{region '#Template'}
	{attribute 'Version' := '1.0.0.0'}
	{attribute 'Tags' := '"LCID": "1031", "Text": "AC, General, night cooling"'}
	{attribute 'Tags' := '"LCID": "1033", "Text": "AC, General, night cooling"'}
	{attribute 'Description' := '"LCID": "1031", "Text": "Nachtkühlung"'}
	{attribute 'Description' := '"LCID": "1033", "Text": "night cooling"'}
{endregion}
FUNCTION_BLOCK FB_BA_AC_SumNgtCol EXTENDS FB_BA_View
VAR_INPUT
	fTRm					: REAL;
	fSpRm					: REAL;
	fTWth					: REAL;		
END_VAR
VAR_OUTPUT
	bQ						: BOOL;
END_VAR
VAR_INPUT CONSTANT
	WthTLoLmt				: FB_BA_AV_Op;	
	RmTHys					: FB_BA_AV_Op;	
	SwiOnDiffT				: FB_BA_AV_Op;	
	SwiOffDiffT				: FB_BA_AV_Op;	
	Q						: FB_BA_BV_Op;																					
	Sched					: FB_BA_SchedM;
END_VAR
VAR
	NgtColFnct				: FB_BA_NgtCol;
END_VAR

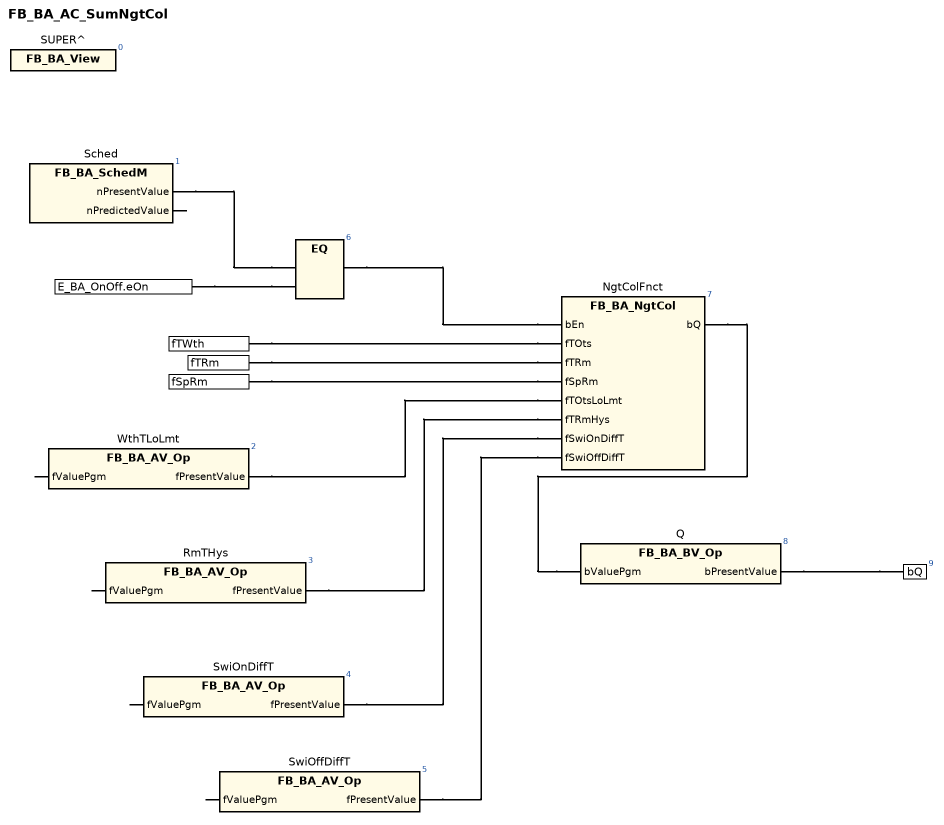
SUPER^(); // FB_BA_View
Sched(); // FB_BA_SchedM
WthTLoLmt(); // FB_BA_AV_Op
RmTHys(); // FB_BA_AV_Op
SwiOnDiffT(); // FB_BA_AV_Op
SwiOffDiffT(); // FB_BA_AV_Op
NgtColFnct(
    bEn := Sched.nPresentValue = E_BA_OnOff.eOn,
    fTOts := fTWth,
    fTRm := fTRm,
    fSpRm := fSpRm,
    fTOtsLoLmt := WthTLoLmt.fPresentValue,
    fTRmHys := RmTHys.fPresentValue,
    fSwiOnDiffT := SwiOnDiffT.fPresentValue,
    fSwiOffDiffT := SwiOffDiffT.fPresentValue); // FB_BA_NgtCol
Q(bValuePgm := NgtColFnct.bQ); // FB_BA_BV_Op
bQ := Q.bPresentValue;

METHOD FB_init : BOOL
VAR_INPUT
	bInitRetains : BOOL; // if TRUE, the retain variables are initialized (warm start / cold start)
	bInCopyCode : BOOL;  // if TRUE, the instance afterwards gets moved into the copy code (online change)
END_VAR
WthTLoLmt.iParent			:= THIS^;
WthTLoLmt.iLabel			:= LblCmpAC.General_SumNgtCol_WthTLoLmt;			
WthTLoLmt.sObjectName		:= '{Idx=01}';								 	 
WthTLoLmt.eUnit				:= E_BA_Unit.eTemperature_DegreesCelsius;  
WthTLoLmt.fValueRm			:= 9.0;

RmTHys.iParent				:= THIS^;
RmTHys.iLabel				:= LblCmpAC.General_SumNgtCol_RmTHys;			
RmTHys.sObjectName			:= '{Idx=01}';								 	 
RmTHys.eUnit				:= E_BA_Unit.eTemperature_DegreesCelsius;  
RmTHys.fValueRm				:= 2.0;

SwiOnDiffT.iParent			:= THIS^;
SwiOnDiffT.iLabel			:= LblCmpAC.General_SumNgtCol_SwiOnDiffT;			
SwiOnDiffT.sObjectName		:= '{Idx=01}';								 	 
SwiOnDiffT.eUnit			:= E_BA_Unit.eTemperature_DegreesCelsius;  
SwiOnDiffT.fValueRm			:= 7.0;

SwiOffDiffT.iParent			:= THIS^;
SwiOffDiffT.iLabel			:= LblCmpAC.General_SumNgtCol_SwiOffDiffT;			
SwiOffDiffT.sObjectName		:= '{Idx=02}';								 	 
SwiOffDiffT.eUnit			:= E_BA_Unit.eTemperature_DegreesCelsius;  
SwiOffDiffT.fValueRm		:= 5.0;

Q.iParent					:= THIS^;
Q.iLabel					:= LblCmpAC.General_SumNgtCol_Q;												 
Q.sObjectName				:= '{Idx=01}';
Q.sInactiveText				:= txtEvent_Off;
Q.sActiveText				:= txtEvent_On;
Q.bValueRm					:= FALSE;								
Q.eToggleMode 				:= E_BA_ToggleMode.eSwitch;

Sched.iParent											:= THIS^;
Sched.iLabel											:= LblCmpAC.General_SumNgtCol_Sched;							
Sched.sObjectName										:= '{Idx=01}';		
Sched.aStateText[1]										:= txtEvent_Off;
Sched.aStateText[2]										:= txtEvent_On;
Sched.nPredictTime										:= 0;
Sched.nDefaultValue										:= E_BA_OnOff.eOff;
Sched.bWriteWeekly										:= FALSE;
//	Monday
Sched.aWeek[E_BA_Weekday.eMonday,1].eState				:= E_BA_SchedEntryState.eValue;
Sched.aWeek[E_BA_Weekday.eMonday,1].uValue.udiVal		:= E_BA_OnOff.eOn;
Sched.aWeek[E_BA_Weekday.eMonday,1].stTime.nHour		:= 1;
Sched.aWeek[E_BA_Weekday.eMonday,1].stTime.nMinute		:= 0;
Sched.aWeek[E_BA_Weekday.eMonday,1].stTime.nSecond		:= 0;
Sched.aWeek[E_BA_Weekday.eMonday,2].eState				:= E_BA_SchedEntryState.eValue;
Sched.aWeek[E_BA_Weekday.eMonday,2].uValue.udiVal		:= E_BA_OnOff.eOff;
Sched.aWeek[E_BA_Weekday.eMonday,2].stTime.nHour		:= 5;
Sched.aWeek[E_BA_Weekday.eMonday,2].stTime.nMinute		:= 0;
Sched.aWeek[E_BA_Weekday.eMonday,2].stTime.nSecond		:= 0;
Sched.aWeek[E_BA_Weekday.eMonday,3].eState				:= E_BA_SchedEntryState.eValue;
Sched.aWeek[E_BA_Weekday.eMonday,3].uValue.udiVal		:= E_BA_OnOff.eOff;
Sched.aWeek[E_BA_Weekday.eMonday,3].stTime.nHour		:= 0;
Sched.aWeek[E_BA_Weekday.eMonday,3].stTime.nMinute		:= 0;
Sched.aWeek[E_BA_Weekday.eMonday,3].stTime.nSecond		:= 0;
//	Tuesday
Sched.aWeek[E_BA_Weekday.eTuesday,1].eState				:= E_BA_SchedEntryState.eValue;
Sched.aWeek[E_BA_Weekday.eTuesday,1].uValue.udiVal		:= E_BA_OnOff.eOn;
Sched.aWeek[E_BA_Weekday.eTuesday,1].stTime.nHour		:= 1;
Sched.aWeek[E_BA_Weekday.eTuesday,1].stTime.nMinute		:= 0;
Sched.aWeek[E_BA_Weekday.eTuesday,1].stTime.nSecond		:= 0;
Sched.aWeek[E_BA_Weekday.eTuesday,2].eState				:= E_BA_SchedEntryState.eValue;
Sched.aWeek[E_BA_Weekday.eTuesday,2].uValue.udiVal		:= E_BA_OnOff.eOff;
Sched.aWeek[E_BA_Weekday.eTuesday,2].stTime.nHour		:= 5;
Sched.aWeek[E_BA_Weekday.eTuesday,2].stTime.nMinute		:= 0;
Sched.aWeek[E_BA_Weekday.eTuesday,2].stTime.nSecond		:= 0;
Sched.aWeek[E_BA_Weekday.eTuesday,3].eState				:= E_BA_SchedEntryState.eValue;
Sched.aWeek[E_BA_Weekday.eTuesday,3].uValue.udiVal		:= E_BA_OnOff.eOff;
Sched.aWeek[E_BA_Weekday.eTuesday,3].stTime.nHour		:= 0;
Sched.aWeek[E_BA_Weekday.eTuesday,3].stTime.nMinute		:= 0;
Sched.aWeek[E_BA_Weekday.eTuesday,3].stTime.nSecond		:= 0;
//	Wednesday
Sched.aWeek[E_BA_Weekday.eWednesday,1].eState			:= E_BA_SchedEntryState.eValue;
Sched.aWeek[E_BA_Weekday.eWednesday,1].uValue.udiVal	:= E_BA_OnOff.eOn;
Sched.aWeek[E_BA_Weekday.eWednesday,1].stTime.nHour		:= 1;
Sched.aWeek[E_BA_Weekday.eWednesday,1].stTime.nMinute	:= 0;
Sched.aWeek[E_BA_Weekday.eWednesday,1].stTime.nSecond	:= 0;
Sched.aWeek[E_BA_Weekday.eWednesday,2].eState			:= E_BA_SchedEntryState.eValue;
Sched.aWeek[E_BA_Weekday.eWednesday,2].uValue.udiVal	:= E_BA_OnOff.eOff;
Sched.aWeek[E_BA_Weekday.eWednesday,2].stTime.nHour		:= 5;
Sched.aWeek[E_BA_Weekday.eWednesday,2].stTime.nMinute	:= 0;
Sched.aWeek[E_BA_Weekday.eWednesday,2].stTime.nSecond	:= 0;
Sched.aWeek[E_BA_Weekday.eWednesday,3].eState			:= E_BA_SchedEntryState.eValue;
Sched.aWeek[E_BA_Weekday.eWednesday,3].uValue.udiVal	:= E_BA_OnOff.eOff;
Sched.aWeek[E_BA_Weekday.eWednesday,3].stTime.nHour		:= 0;
Sched.aWeek[E_BA_Weekday.eWednesday,3].stTime.nMinute	:= 0;
Sched.aWeek[E_BA_Weekday.eWednesday,3].stTime.nSecond	:= 0;
//	Thursday
Sched.aWeek[E_BA_Weekday.eThursday,1].eState			:= E_BA_SchedEntryState.eValue;
Sched.aWeek[E_BA_Weekday.eThursday,1].uValue.udiVal		:= E_BA_OnOff.eOn;
Sched.aWeek[E_BA_Weekday.eThursday,1].stTime.nHour		:= 1;
Sched.aWeek[E_BA_Weekday.eThursday,1].stTime.nMinute	:= 0;
Sched.aWeek[E_BA_Weekday.eThursday,1].stTime.nSecond	:= 0;
Sched.aWeek[E_BA_Weekday.eThursday,2].eState			:= E_BA_SchedEntryState.eValue;
Sched.aWeek[E_BA_Weekday.eThursday,2].uValue.udiVal		:= E_BA_OnOff.eOff;
Sched.aWeek[E_BA_Weekday.eThursday,2].stTime.nHour		:= 5;
Sched.aWeek[E_BA_Weekday.eThursday,2].stTime.nMinute	:= 0;
Sched.aWeek[E_BA_Weekday.eThursday,2].stTime.nSecond	:= 0;
Sched.aWeek[E_BA_Weekday.eThursday,3].eState			:= E_BA_SchedEntryState.eValue;
Sched.aWeek[E_BA_Weekday.eThursday,3].uValue.udiVal		:= E_BA_OnOff.eOff;
Sched.aWeek[E_BA_Weekday.eThursday,3].stTime.nHour		:= 0;
Sched.aWeek[E_BA_Weekday.eThursday,3].stTime.nMinute	:= 0;
Sched.aWeek[E_BA_Weekday.eThursday,3].stTime.nSecond	:= 0;
//	Friday
Sched.aWeek[E_BA_Weekday.eFriday,1].eState				:= E_BA_SchedEntryState.eValue;
Sched.aWeek[E_BA_Weekday.eFriday,1].uValue.udiVal		:= E_BA_OnOff.eOn;
Sched.aWeek[E_BA_Weekday.eFriday,1].stTime.nHour		:= 1;
Sched.aWeek[E_BA_Weekday.eFriday,1].stTime.nMinute		:= 0;
Sched.aWeek[E_BA_Weekday.eFriday,1].stTime.nSecond		:= 0;
Sched.aWeek[E_BA_Weekday.eFriday,2].eState				:= E_BA_SchedEntryState.eValue;
Sched.aWeek[E_BA_Weekday.eFriday,2].uValue.udiVal		:= E_BA_OnOff.eOff;
Sched.aWeek[E_BA_Weekday.eFriday,2].stTime.nHour		:= 5;
Sched.aWeek[E_BA_Weekday.eFriday,2].stTime.nMinute		:= 0;
Sched.aWeek[E_BA_Weekday.eFriday,2].stTime.nSecond		:= 0;
Sched.aWeek[E_BA_Weekday.eFriday,3].eState				:= E_BA_SchedEntryState.eValue;
Sched.aWeek[E_BA_Weekday.eFriday,3].uValue.udiVal		:= E_BA_OnOff.eOff;
Sched.aWeek[E_BA_Weekday.eFriday,3].stTime.nHour		:= 0;
Sched.aWeek[E_BA_Weekday.eFriday,3].stTime.nMinute		:= 0;
Sched.aWeek[E_BA_Weekday.eFriday,3].stTime.nSecond		:= 0;
Sched.bWriteException									:= FALSE;
END_METHOD

END_FUNCTION_BLOCK

(* stored: Version 1.1.0.1, ProductVersion 3.1.4024.9
   POU FB_BA_AC_SumNgtCol: Id {b7a72e16-6429-436a-8468-b71e16e0326a}, SpecialFunc None
   Method FB_init: Id {8f29484c-1e67-4db5-bcf9-5c1003f07352} *)
